(* PLC project Unnamed, Unknown Unnamed 1 *)
(* stored: creationDateTime 2024-03-06T23:19:10, modificationDateTime 2024-03-08T11:47:02 *)

PROGRAM program0
  VAR
    SPD AT %IX0.4 : BOOL;
  END_VAR
  VAR
    STOP1 : BOOL;
    STOP2 : BOOL;
    STOP3 : BOOL;
    JFD_OUT : BOOL;
  END_VAR
  VAR
    JFD AT %IX0.2 : BOOL;
    JFD_RR AT %QX0.2 : BOOL;
  END_VAR
  VAR
    JFD_SPD : INT := 0;
    A1 : BOOL := 1;
    A2 : BOOL := 1;
  END_VAR
  VAR
    DRON AT %IX0.3 : BOOL;
  END_VAR
  VAR
    TON0 : TON;
  END_VAR
  VAR
    JRV AT %IX0.1 : BOOL;
    JRV_RR AT %QX0.1 : BOOL;
  END_VAR
  VAR
    TON1 : TON;
    JRV_OUT : BOOL;
    JRV_SPD : INT;
  END_VAR
  VAR
    RUN AT %IX0.0 : BOOL;
  END_VAR
  VAR
    RUN_RR : BOOL;
  END_VAR
  VAR
    RUN_OUT AT %QX0.0 : BOOL;
  END_VAR
  VAR
    TON2 : TON;
    RUN_SPD : INT;
    STOP : BOOL;
  END_VAR
  VAR  (* added by the conversion: wires and edge detectors of the diagram *)
    _BOOL_TO_INT22_OUT : INT;
  END_VAR

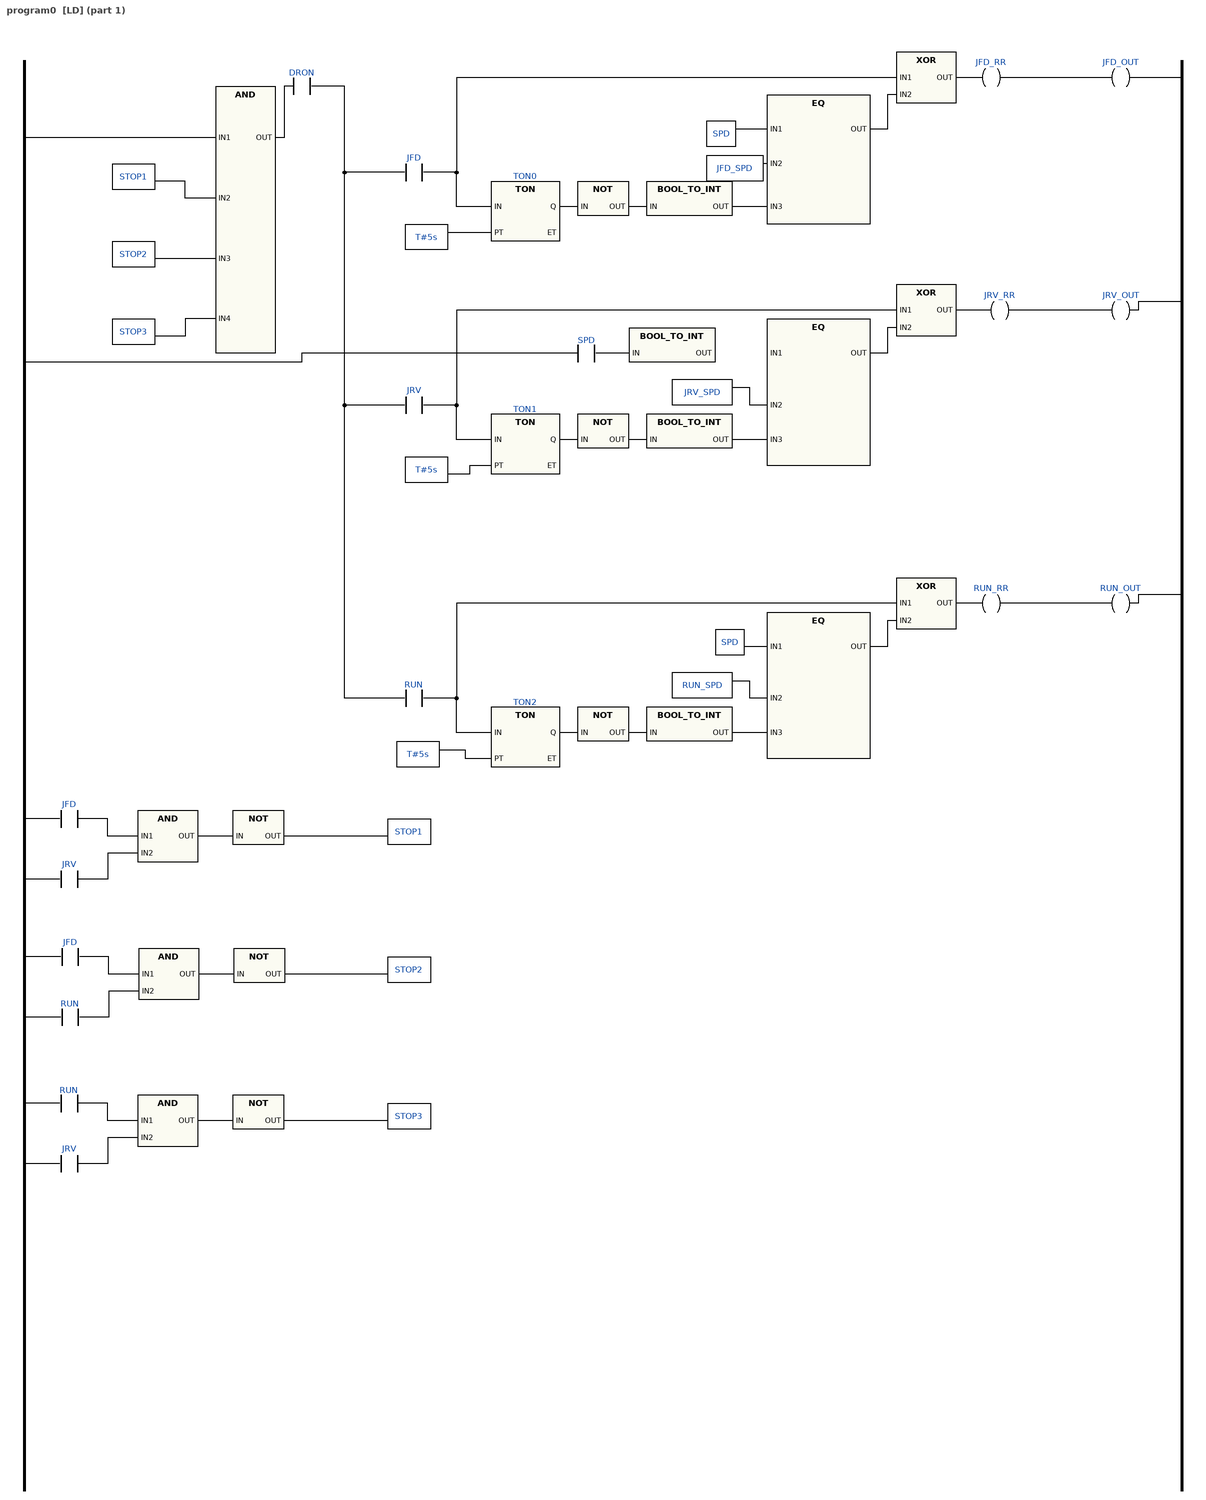
(* LD diagram, written out as Structured Text *)
TON0(IN := TRUE AND STOP1 AND STOP2 AND STOP3 AND DRON AND JFD, PT := T#5s);
JFD_RR := TRUE AND STOP1 AND STOP2 AND STOP3 AND DRON AND JFD XOR EQ(SPD, JFD_SPD, BOOL_TO_INT(NOT TON0.Q));
JFD_OUT := TRUE AND STOP1 AND STOP2 AND STOP3 AND DRON AND JFD XOR EQ(SPD, JFD_SPD, BOOL_TO_INT(NOT TON0.Q));
TON1(IN := TRUE AND STOP1 AND STOP2 AND STOP3 AND DRON AND JRV, PT := T#5s);
JRV_RR := TRUE AND STOP1 AND STOP2 AND STOP3 AND DRON AND JRV XOR EQ(IN2 := JRV_SPD, IN3 := BOOL_TO_INT(NOT TON1.Q));
JRV_OUT := TRUE AND STOP1 AND STOP2 AND STOP3 AND DRON AND JRV XOR EQ(IN2 := JRV_SPD, IN3 := BOOL_TO_INT(NOT TON1.Q));
TON2(IN := TRUE AND STOP1 AND STOP2 AND STOP3 AND DRON AND RUN, PT := T#5s);
RUN_RR := TRUE AND STOP1 AND STOP2 AND STOP3 AND DRON AND RUN XOR EQ(SPD, RUN_SPD, BOOL_TO_INT(NOT TON2.Q));
RUN_OUT := TRUE AND STOP1 AND STOP2 AND STOP3 AND DRON AND RUN XOR EQ(SPD, RUN_SPD, BOOL_TO_INT(NOT TON2.Q));
STOP1 := NOT (JFD AND JRV);
STOP2 := NOT (JFD AND RUN);
STOP3 := NOT (RUN AND JRV);
_BOOL_TO_INT22_OUT := BOOL_TO_INT(SPD);
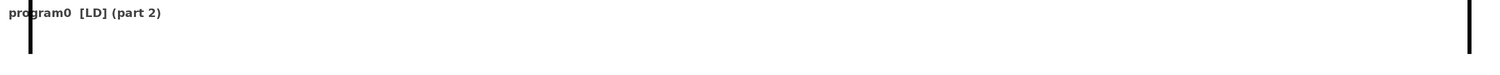
END_PROGRAM

CONFIGURATION Config0
  RESOURCE Res0 ON PLC
    TASK task0(INTERVAL := T#20ms, PRIORITY := 0);
    PROGRAM instance0 WITH task0 : program0;
  END_RESOURCE
END_CONFIGURATION
